% RSLogix 500 project traffic signal.RSS, saved by version 8.30.00.16 %
PROJECT "UNTITLED"    % processor: Bul.1763 MicroLogix 1100 Series B %

PROGRAM FILES
  LAD 2   6 rungs

DATA FILES
  O0 OUTPUT  4 elements
  I1 INPUT  6 elements
  S2 STATUS  66 elements
  B3 BINARY  1 elements
  T4 TIMER  3 elements
  C5 COUNTER  1 elements
  R6 CONTROL  1 elements
  N7 INTEGER  1 elements
  F8 FLOAT  1 elements

LADDER 2
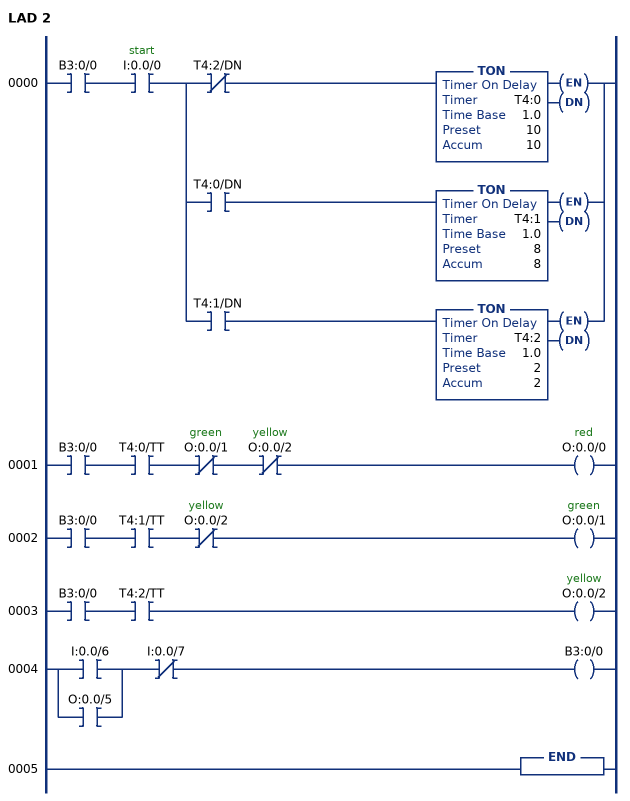
% Rung: 0 %
SOR XIC B3:0/0 XIC I:0.0/0 BST XIO T4:2/DN TON T4:0 1.0 10 10 NXB BST XIC T4:0/DN TON T4:1 1.0 8 8 NXB XIC T4:1/DN TON T4:2 1.0 2 2 BND BND EOR
%   I:0.0/0  "start" %
% Rung: 1 %
SOR XIC B3:0/0 XIC T4:0/TT XIO O:0.0/1 XIO O:0.0/2 OTE O:0.0/0 EOR
%   O:0.0/1  "green" %
%   O:0.0/2  "yellow" %
%   O:0.0/0  "red" %
% Rung: 2 %
SOR XIC B3:0/0 XIC T4:1/TT XIO O:0.0/2 OTE O:0.0/1 EOR
%   O:0.0/2  "yellow" %
%   O:0.0/1  "green" %
% Rung: 3 %
SOR XIC B3:0/0 XIC T4:2/TT OTE O:0.0/2 EOR
%   O:0.0/2  "yellow" %
% Rung: 4 %
SOR BST XIC I:0.0/6 NXB XIC O:0.0/5 BND XIO I:0.0/7 OTE B3:0/0 EOR
% Rung: 5 %
SOR END EOR

DATA TABLE (non-zero values as saved)
DATA T4
% .PRE .ACC %
% T4:0 % 10 10
% T4:1 % 8 8
% T4:2 % 2 2
